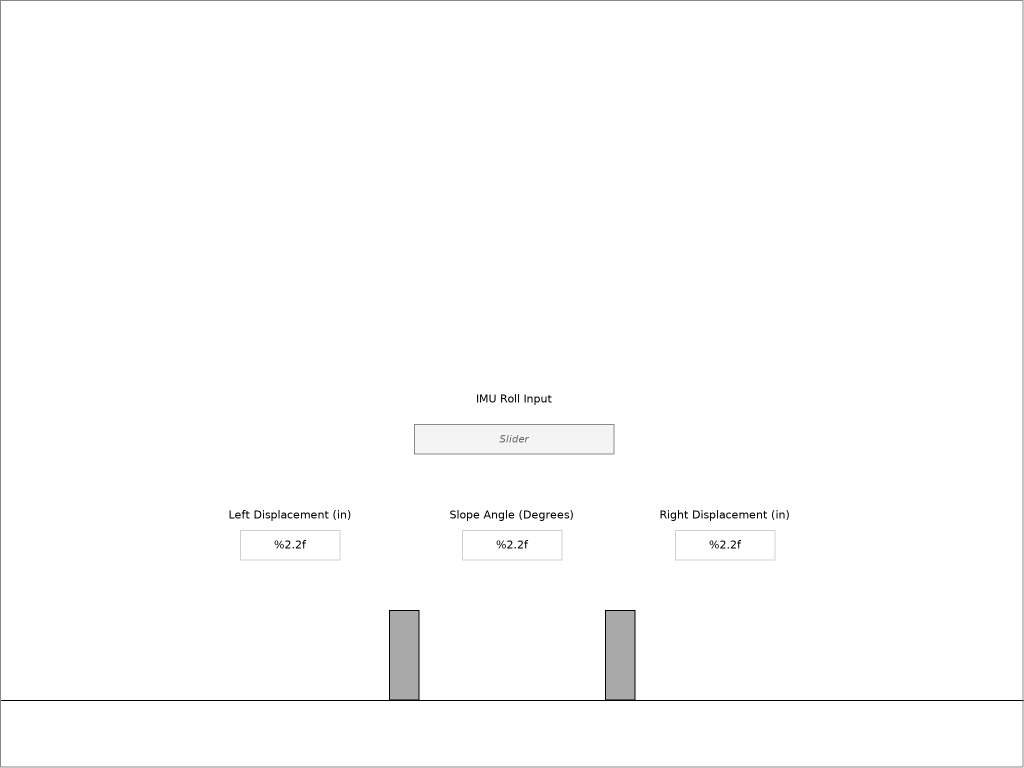
VISUALIZATION TiltControlTest  // 1024x768
    Line (0,700) (1024,700)
        p2858320360: HARV.TiltControl.SlopeAngle
        p2738717112: (HARV.TiltControl.TiltDisplacement * 3) / 2
    Rectangle (389,610 30x90)
        p2738717112: HARV.TiltControl.TiltLeftDisplacement *3
    Rectangle (605,610 30x90)
        p2738717112: HARV.TiltControl.TiltRightDisplacement * 3
    Group (437,500 150x60)
        Textfield (25,30 100x30), "%2.2f", text variable: HARV.TiltControl.SlopeAngle
            OnMouseClick: write the text variable via Default, min -10, max 10
        Label (0,0 150x30), "Slope Angle (Degrees)"
    Group (650,500 150x60)
        Textfield (25,30 100x30), "%2.2f", text variable: HARV.TiltControl.TiltRightDisplacement
            OnMouseClick: write the text variable via Default, min -10, max 10
        Label (0,0 150x30), "Right Displacement (in)"
    Group (215,500 150x60)
        Textfield (25,30 100x30), "%2.2f", text variable: HARV.TiltControl.TiltLeftDisplacement
            OnMouseClick: write the text variable via Default, min -10, max 10
        Label (0,0 150x30), "Left Displacement (in)"
    Slider (414,424 200x30), variable: HARV.TiltControl.IMU_Roll, scale -11..11
    Label (439,384 150x30), "IMU Roll Input"
END_VISUALIZATION

(* stored: Version 1.1.0.1, ProductVersion 3.1.4024.12
   Visu TiltControlTest: Id {a0f1d7e1-41a9-42ef-a039-38385dcd58fd} *)
